(* IEC 61131-3 sources: plcc/crates/plcc-stdlib/st, 4 files *)

(* ---- bistable.st ---- *)
(* SPDX-License-Identifier: MPL-2.0 *)
(*
 * IEC 61131-3 section 2.5.2.2 — bistable elements.
 *
 * The bodies below are the standard's own ST definitions.
 *)

(* SR — SET-dominant bistable.
 * When S1 and R are both TRUE, Q1 is TRUE. *)
FUNCTION_BLOCK SR
VAR_INPUT
    S1 : BOOL;
    R : BOOL;
END_VAR
VAR_OUTPUT
    Q1 : BOOL;
END_VAR
    Q1 := S1 OR (NOT R AND Q1);
END_FUNCTION_BLOCK

(* RS — RESET-dominant bistable.
 * When S and R1 are both TRUE, Q1 is FALSE. *)
FUNCTION_BLOCK RS
VAR_INPUT
    S : BOOL;
    R1 : BOOL;
END_VAR
VAR_OUTPUT
    Q1 : BOOL;
END_VAR
    Q1 := NOT R1 AND (S OR Q1);
END_FUNCTION_BLOCK

(* ---- counters.st ---- *)
(* SPDX-License-Identifier: MPL-2.0 *)
(*
 * IEC 61131-3 section 2.5.2.3.3 — counters.
 *
 * The standard declares the count inputs as `CU : BOOL R_EDGE`, i.e. the
 * counting inputs are edge-triggered. That declaration form is expressed here
 * with an explicit edge memory, which is exactly equivalent and does not rely
 * on R_EDGE support in the front end.
 *
 * CV saturates at the limits of INT. It does NOT wrap: the standard guards the
 * increment with `CV < PVmax` and the decrement with `CV > PVmin`.
 *)

(* CTU — up counter.
 * R has priority over CU. Q := (CV >= PV). *)
FUNCTION_BLOCK CTU
VAR_INPUT
    CU : BOOL;
    R : BOOL;
    PV : INT;
END_VAR
VAR_OUTPUT
    Q : BOOL;
    CV : INT;
END_VAR
VAR
    M_CU : BOOL := FALSE;
    CU_EDGE : BOOL;
END_VAR
    CU_EDGE := CU AND NOT M_CU;
    M_CU := CU;
    IF R THEN
        CV := 0;
    ELSIF CU_EDGE THEN
        IF CV < 32767 THEN
            CV := CV + 1;
        END_IF;
    END_IF;
    Q := CV >= PV;
END_FUNCTION_BLOCK

(* CTD — down counter.
 * LD has priority over CD and loads CV := PV. Q := (CV <= 0). *)
FUNCTION_BLOCK CTD
VAR_INPUT
    CD : BOOL;
    LD : BOOL;
    PV : INT;
END_VAR
VAR_OUTPUT
    Q : BOOL;
    CV : INT;
END_VAR
VAR
    M_CD : BOOL := FALSE;
    CD_EDGE : BOOL;
END_VAR
    CD_EDGE := CD AND NOT M_CD;
    M_CD := CD;
    IF LD THEN
        CV := PV;
    ELSIF CD_EDGE THEN
        IF CV > -32768 THEN
            CV := CV - 1;
        END_IF;
    END_IF;
    Q := CV <= 0;
END_FUNCTION_BLOCK

(* CTUD — up/down counter.
 *
 * Precedence, per the standard's body:
 *   R dominates LD, and both dominate counting.
 *   When CU and CD are edge-active in the same scan, CV does NOT change.
 *
 * QU := (CV >= PV);  QD := (CV <= 0). *)
FUNCTION_BLOCK CTUD
VAR_INPUT
    CU : BOOL;
    CD : BOOL;
    R : BOOL;
    LD : BOOL;
    PV : INT;
END_VAR
VAR_OUTPUT
    QU : BOOL;
    QD : BOOL;
    CV : INT;
END_VAR
VAR
    M_CU : BOOL := FALSE;
    M_CD : BOOL := FALSE;
    CU_EDGE : BOOL;
    CD_EDGE : BOOL;
    BOTH : BOOL;
END_VAR
    CU_EDGE := CU AND NOT M_CU;
    CD_EDGE := CD AND NOT M_CD;
    M_CU := CU;
    M_CD := CD;
    BOTH := CU_EDGE AND CD_EDGE;
    IF R THEN
        CV := 0;
    ELSIF LD THEN
        CV := PV;
    ELSIF NOT BOTH THEN
        IF CU_EDGE THEN
            IF CV < 32767 THEN
                CV := CV + 1;
            END_IF;
        ELSIF CD_EDGE THEN
            IF CV > -32768 THEN
                CV := CV - 1;
            END_IF;
        END_IF;
    END_IF;
    QU := CV >= PV;
    QD := CV <= 0;
END_FUNCTION_BLOCK

(* ---- edge.st ---- *)
(* SPDX-License-Identifier: MPL-2.0 *)
(*
 * IEC 61131-3 section 2.5.2.3 — edge detection.
 *
 * The bodies below are the standard's own ST definitions, including the
 * asymmetric initial value of the edge memory: R_TRIG's M starts FALSE, so a
 * CLK that is already TRUE on the first call produces a pulse; F_TRIG's M
 * starts TRUE, so a CLK that is already FALSE on the first call does not.
 *)

(* R_TRIG — rising edge detector.
 * Q is TRUE for exactly one scan following a FALSE -> TRUE transition of CLK. *)
FUNCTION_BLOCK R_TRIG
VAR_INPUT
    CLK : BOOL;
END_VAR
VAR_OUTPUT
    Q : BOOL;
END_VAR
VAR
    M : BOOL := FALSE;
END_VAR
    Q := CLK AND NOT M;
    M := CLK;
END_FUNCTION_BLOCK

(* F_TRIG — falling edge detector.
 * Q is TRUE for exactly one scan following a TRUE -> FALSE transition of CLK. *)
FUNCTION_BLOCK F_TRIG
VAR_INPUT
    CLK : BOOL;
END_VAR
VAR_OUTPUT
    Q : BOOL;
END_VAR
VAR
    M : BOOL := TRUE;
END_VAR
    Q := NOT CLK AND NOT M;
    M := NOT CLK;
END_FUNCTION_BLOCK

(* ---- timers.st ---- *)
(* SPDX-License-Identifier: MPL-2.0 *)
(*
 * IEC 61131-3 section 2.5.2.4 — timers.
 *
 * These read the platform clock through MONOTONIC_NS(), which compiles to a
 * call to the external `plcc_monotonic_ns() -> LINT` symbol. Elapsed time is
 * therefore measured against real time, not counted in scans, so timing does
 * not drift with scan period. See docs/runtime-symbols.md.
 *
 * TIME and LTIME are laid out as signed 64-bit nanoseconds, which is what
 * MONOTONIC_NS() returns, so the clock readings are kept as TIME and no
 * conversion is needed anywhere below.
 *)

(* TON — on-delay timer.
 *   Q goes TRUE after IN has been continuously TRUE for PT.
 *   ET counts up from 0 and is capped at PT, where it freezes.
 *   IN going FALSE resets Q and ET immediately. *)
FUNCTION_BLOCK TON
VAR_INPUT
    IN : BOOL;
    PT : TIME;
END_VAR
VAR_OUTPUT
    Q : BOOL;
    ET : TIME;
END_VAR
VAR
    RUNNING : BOOL := FALSE;
    START_NS : TIME;
    NOW_NS : TIME;
    ELAPSED : TIME;
END_VAR
    NOW_NS := MONOTONIC_NS();
    IF IN THEN
        IF NOT RUNNING THEN
            RUNNING := TRUE;
            START_NS := NOW_NS;
        END_IF;
        ELAPSED := NOW_NS - START_NS;
        IF ELAPSED >= PT THEN
            ET := PT;
            Q := TRUE;
        ELSE
            ET := ELAPSED;
            Q := FALSE;
        END_IF;
    ELSE
        RUNNING := FALSE;
        ET := T#0s;
        Q := FALSE;
    END_IF;
END_FUNCTION_BLOCK

(* TOF — off-delay timer. The mirror of TON.
 *   Q goes TRUE immediately when IN goes TRUE.
 *   On the falling edge of IN, ET counts up from 0; when it reaches PT, Q goes
 *   FALSE and ET freezes at PT.
 *   IN going TRUE again clears ET and cancels the off-delay. *)
FUNCTION_BLOCK TOF
VAR_INPUT
    IN : BOOL;
    PT : TIME;
END_VAR
VAR_OUTPUT
    Q : BOOL;
    ET : TIME;
END_VAR
VAR
    PREV_IN : BOOL := FALSE;
    RUNNING : BOOL := FALSE;
    START_NS : TIME;
    NOW_NS : TIME;
    ELAPSED : TIME;
END_VAR
    NOW_NS := MONOTONIC_NS();
    IF IN THEN
        RUNNING := FALSE;
        ET := T#0s;
        Q := TRUE;
    ELSE
        IF PREV_IN THEN
            RUNNING := TRUE;
            START_NS := NOW_NS;
        END_IF;
        IF RUNNING THEN
            ELAPSED := NOW_NS - START_NS;
            IF ELAPSED >= PT THEN
                ET := PT;
                Q := FALSE;
                RUNNING := FALSE;
            ELSE
                ET := ELAPSED;
                Q := TRUE;
            END_IF;
        END_IF;
    END_IF;
    PREV_IN := IN;
END_FUNCTION_BLOCK

(* TP — pulse timer.
 *   A rising edge of IN starts a pulse of length PT: Q is TRUE and ET counts up.
 *   The pulse is NOT retriggerable — further rising edges of IN while the pulse
 *   is running are ignored, and ET is not restarted.
 *   When the pulse ends, Q goes FALSE and ET holds at PT until IN goes FALSE. *)
FUNCTION_BLOCK TP
VAR_INPUT
    IN : BOOL;
    PT : TIME;
END_VAR
VAR_OUTPUT
    Q : BOOL;
    ET : TIME;
END_VAR
VAR
    PREV_IN : BOOL := FALSE;
    RUNNING : BOOL := FALSE;
    START_NS : TIME;
    NOW_NS : TIME;
    ELAPSED : TIME;
    IN_EDGE : BOOL;
END_VAR
    NOW_NS := MONOTONIC_NS();
    IN_EDGE := IN AND NOT PREV_IN;
    PREV_IN := IN;
    IF IN_EDGE THEN
        IF NOT RUNNING THEN
            RUNNING := TRUE;
            START_NS := NOW_NS;
        END_IF;
    END_IF;
    IF RUNNING THEN
        ELAPSED := NOW_NS - START_NS;
        IF ELAPSED >= PT THEN
            ET := PT;
            Q := FALSE;
            RUNNING := FALSE;
        ELSE
            ET := ELAPSED;
            Q := TRUE;
        END_IF;
    ELSE
        Q := FALSE;
        IF NOT IN THEN
            ET := T#0s;
        END_IF;
    END_IF;
END_FUNCTION_BLOCK

(* RTO — retentive on-delay timer. Not an IEC 61131-3 standard FB: plcc's IEC
 * counterpart of the Logix RTO instruction (1756-RM003 "Retentive Timer On"),
 * so ladder translated from Logix keeps its meaning (docs/ladder-translation.md).
 *   ET accumulates while IN is TRUE and holds its value while IN is FALSE.
 *   Q := ET >= PT; ET stops at PT (Logix: accumulation stops once DN is set).
 *   R clears ET and Q (Logix: the RES instruction). *)
FUNCTION_BLOCK RTO
VAR_INPUT
    IN : BOOL;
    R : BOOL;
    PT : TIME;
END_VAR
VAR_OUTPUT
    Q : BOOL;
    ET : TIME;
END_VAR
VAR
    RUNNING : BOOL := FALSE;
    LAST_NS : TIME;
    NOW_NS : TIME;
END_VAR
    NOW_NS := MONOTONIC_NS();
    IF R THEN
        ET := T#0s;
        RUNNING := FALSE;
    ELSIF IN THEN
        IF RUNNING AND ET < PT THEN
            ET := ET + (NOW_NS - LAST_NS);
            IF ET > PT THEN
                ET := PT;
            END_IF;
        END_IF;
        RUNNING := TRUE;
        LAST_NS := NOW_NS;
    ELSE
        RUNNING := FALSE;
    END_IF;
    Q := ET >= PT AND NOT R;
END_FUNCTION_BLOCK
